LIN {X 0,Y 81.498,Z 212.955,A -85,B 0,C 180,E1 -29781.837,E2 -29781.837} C_VEL
LIN {X 0,Y 84.954,Z 223.328,A -85,B 0,C 180,E1 -29789.059,E2 -29789.059} C_VEL
LIN {X 0,Y 88.345,Z 233.499,A -85,B 0,C 180,E1 -29794.807,E2 -29794.807} C_VEL
LIN {X 0,Y 92.972,Z 247.732,A -85,B 0,C 180,E1 -29801.381,E2 -29801.381} C_VEL
LIN {X 0,Y 75.771,Z 322.387,A -85,B 0,C 180,E1 -29809.104,E2 -29809.104} C_VEL
LIN {X 0,Y 70.598,Z 340.758,A -85,B 0,C 180,E1 -29812.018,E2 -29812.018} C_VEL
LIN {X 0,Y 64.901,Z 358.077,A -85,B 0,C 180,E1 -29815.953,E2 -29815.953} C_VEL
LIN {X 0,Y 57.963,Z 376.296,A -85,B 0,C 180,E1 -29821.924,E2 -29821.924} C_VEL
LIN {X 0,Y 50.843,Z 393.773,A -85,B 0,C 180,E1 -29830.512,E2 -29830.512} C_VEL
LIN {X 0,Y 44.399,Z 410.254,A -85,B 0,C 180,E1 -29843.006,E2 -29843.006} C_VEL
LIN {X 0,Y 40.062,Z 424.851,A -85,B 0,C 180,E1 -29859.459,E2 -29859.459} C_VEL
LIN {X 0,Y 38.918,Z 435.167,A -85,B 0,C 180,E1 -29874.818,E2 -29874.818} C_VEL
LIN {X 0,Y 40.086,Z 444.149,A -85,B 0,C 180,E1 -29890.096,E2 -29890.096} C_VEL
LIN {X 0,Y 42.987,Z 451.752,A -85,B 0,C 180,E1 -29904.124,E2 -29904.124} C_VEL
LIN {X 0,Y 48.332,Z 459.273,A -85,B 0,C 180,E1 -29918.169,E2 -29918.169} C_VEL
LIN {X 0,Y 52.134,Z 462.9,A -85,B 0,C 180,E1 -29924.447,E2 -29924.447} C_VEL
LIN {X 0,Y 51.741,Z 462.795,A -85,B 0,C 180,E1 -29927.216,E2 -29927.216} C_VEL
LIN {X 0,Y 46.77,Z 457.154,A -85,B 0,C 180,E1 -29947.357,E2 -29947.357} C_VEL
LIN {X 0,Y 46.468,Z 455.688,A -85,B 0,C 180,E1 -29952.387,E2 -29952.387} C_VEL
LIN {X 0,Y 46.065,Z 453.922,A -85,B 0,C 180,E1 -29956.765,E2 -29956.765} C_VEL
LIN {X 0,Y 43.68,Z 447.526,A -85,B 0,C 180,E1 -29967.689,E2 -29967.689} C_VEL
LIN {X 0,Y 42.428,Z 436.729,A -85,B 0,C 180,E1 -29984.38,E2 -29984.38} C_VEL
LIN {X 0,Y 44.138,Z 425.938,A -85,B 0,C 180,E1 -29998.527,E2 -29998.527} C_VEL
LIN {X 0,Y 48.424,Z 412.157,A -85,B 0,C 180,E1 -30012.045,E2 -30012.045} C_VEL
LIN {X 0,Y 54.366,Z 397.007,A -85,B 0,C 180,E1 -30022.345,E2 -30022.345} C_VEL
LIN {X 0,Y 60.976,Z 380.581,A -85,B 0,C 180,E1 -30029.81,E2 -30029.81} C_VEL
LIN {X 0,Y 67.321,Z 363.42,A -85,B 0,C 180,E1 -30035.134,E2 -30035.134} C_VEL
LIN {X 0,Y 73.035,Z 346.162,A -85,B 0,C 180,E1 -30038.771,E2 -30038.771} C_VEL
LIN {X 0,Y 77.413,Z 329.485,A -85,B 0,C 180,E1 -30041.354,E2 -30041.354} C_VEL
LIN {X 0,Y 94.399,Z 256.118,A -85,B 0,C 180,E1 -30049.009,E2 -30049.009} C_VEL
LIN {X 0,Y 89.802,Z 238.607,A -85,B 0,C 180,E1 -30055.909,E2 -30055.909} C_VEL
LIN {X 0,Y 87.812,Z 231.246,A -85,B 0,C 180,E1 -30059.302,E2 -30059.302} C_VEL
LIN {X 0,Y 83.874,Z 219.706,A -85,B 0,C 180,E1 -30066.271,E2 -30066.271} C_VEL
LIN {X 0,Y 81.116,Z 211.549,A -85,B 0,C 180,E1 -30072.319,E2 -30072.319} C_VEL
LIN {X 0,Y 79.343,Z 206.703,A -85,B 0,C 180,E1 -30076.883,E2 -30076.883} C_VEL
LIN {X 0,Y 77.372,Z 202.569,A -85,B 0,C 180,E1 -30082.396,E2 -30082.396} C_VEL
LIN {X 0,Y 76.416,Z 200.778,A -85,B 0,C 180,E1 -30085.579,E2 -30085.579} C_VEL
LIN {X 0,Y 75.225,Z 198.037,A -85,B 0,C 180,E1 -30090.911,E2 -30090.911} C_VEL
LIN {X 0,Y 73.855,Z 194.358,A -85,B 0,C 180,E1 -30105.053,E2 -30105.053} C_VEL
LIN {X 0,Y 73.889,Z 194.326,A -85,B 0,C 180,E1 -30108.716,E2 -30108.716} C_VEL
LIN {X 0,Y 75.492,Z 198.537,A -85,B 0,C 180,E1 -30123.535,E2 -30123.535} C_VEL
LIN {X 0,Y 77.1,Z 201.774,A -85,B 0,C 180,E1 -30129.721,E2 -30129.721} C_VEL
LIN {X 0,Y 78.057,Z 203.875,A -85,B 0,C 180,E1 -30132.788,E2 -30132.788} C_VEL
LIN {X 0,Y 78.673,Z 206.225,A -85,B 0,C 180,E1 -30135,E2 -30135} C_VEL
LIN {X 0,Y 78.846,Z 209.414,A -85,B 0,C 180,E1 -30136.71,E2 -30136.71} C_VEL
LIN {X 0,Y 78.721,Z 219.635,A -85,B 0,C 180,E1 -30140.842,E2 -30140.842} C_VEL
LIN {X 0,Y 78.953,Z 221.239,A -85,B 0,C 180,E1 -30141.776,E2 -30141.776} C_VEL
LIN {X 0,Y 82.123,Z 231.652,A -85,B 0,C 180,E1 -30148.911,E2 -30148.911} C_VEL
LIN {X 0,Y 85.803,Z 243.983,A -85,B 0,C 180,E1 -30155.622,E2 -30155.622} C_VEL
LIN {X 0,Y 87.566,Z 249.754,A -85,B 0,C 180,E1 -30158.369,E2 -30158.369} C_VEL
LIN {X 0,Y 69.671,Z 323.884,A -85,B 0,C 180,E1 -30165.958,E2 -30165.958} C_VEL
LIN {X 0,Y 63.877,Z 343.313,A -85,B 0,C 180,E1 -30169.187,E2 -30169.187} C_VEL
LIN {X 0,Y 57.497,Z 361.158,A -85,B 0,C 180,E1 -30173.543,E2 -30173.543} C_VEL
LIN {X 0,Y 50.547,Z 378.063,A -85,B 0,C 180,E1 -30179.658,E2 -30179.658} C_VEL
LIN {X 0,Y 43.158,Z 395.148,A -85,B 0,C 180,E1 -30189.332,E2 -30189.332} C_VEL
LIN {X 0,Y 37.164,Z 409.779,A -85,B 0,C 180,E1 -30202.431,E2 -30202.431} C_VEL
LIN {X 0,Y 33.075,Z 423.75,A -85,B 0,C 180,E1 -30221.413,E2 -30221.413} C_VEL
LIN {X 0,Y 32.512,Z 434.151,A -85,B 0,C 180,E1 -30239.999,E2 -30239.999} C_VEL
LIN {X 0,Y 34.7,Z 443.052,A -85,B 0,C 180,E1 -30257.685,E2 -30257.685} C_VEL
LIN {X 0,Y 38.033,Z 449.406,A -85,B 0,C 180,E1 -30270.54,E2 -30270.54} C_VEL
LIN {X 0,Y 44.578,Z 457.016,A -85,B 0,C 180,E1 -30285.189,E2 -30285.189} C_VEL
LIN {X 0,Y 44.148,Z 456.848,A -85,B 0,C 180,E1 -30290.441,E2 -30290.441} C_VEL
LIN {X 0,Y 40.851,Z 451.711,A -85,B 0,C 180,E1 -30309.867,E2 -30309.867} C_VEL
LIN {X 0,Y 40.524,Z 450.826,A -85,B 0,C 180,E1 -30312.325,E2 -30312.325} C_VEL
LIN {X 0,Y 37.539,Z 444.264,A -85,B 0,C 180,E1 -30324.622,E2 -30324.622} C_VEL
LIN {X 0,Y 35.942,Z 433.295,A -85,B 0,C 180,E1 -30343.849,E2 -30343.849} C_VEL
LIN {X 0,Y 37.796,Z 421.958,A -85,B 0,C 180,E1 -30360.746,E2 -30360.746} C_VEL
LIN {X 0,Y 42.454,Z 408.36,A -85,B 0,C 180,E1 -30375.478,E2 -30375.478} C_VEL
LIN {X 0,Y 48.556,Z 393.763,A -85,B 0,C 180,E1 -30385.949,E2 -30385.949} C_VEL
LIN {X 0,Y 55.792,Z 376.675,A -85,B 0,C 180,E1 -30393.824,E2 -30393.824} C_VEL
LIN {X 0,Y 62.443,Z 359.243,A -85,B 0,C 180,E1 -30399.052,E2 -30399.052} C_VEL
LIN {X 0,Y 68.54,Z 340.751,A -85,B 0,C 180,E1 -30402.711,E2 -30402.711} C_VEL
LIN {X 0,Y 73.894,Z 319.765,A -85,B 0,C 180,E1 -30405.662,E2 -30405.662} C_VEL
LIN {X 0,Y 88.85,Z 257.627,A -85,B 0,C 180,E1 -30411.928,E2 -30411.928} C_VEL
LIN {X 0,Y 84.552,Z 239.719,A -85,B 0,C 180,E1 -30419.612,E2 -30419.612} C_VEL
LIN {X 0,Y 82.874,Z 233.486,A -85,B 0,C 180,E1 -30422.934,E2 -30422.934} C_VEL
LIN {X 0,Y 79.607,Z 222.985,A -85,B 0,C 180,E1 -30429.922,E2 -30429.922} C_VEL
LIN {X 0,Y 77.751,Z 216.749,A -85,B 0,C 180,E1 -30434.853,E2 -30434.853} C_VEL
LIN {X 0,Y 76.283,Z 212.249,A -85,B 0,C 180,E1 -30439.302,E2 -30439.302} C_VEL
LIN {X 0,Y 74.59,Z 208.154,A -85,B 0,C 180,E1 -30445.095,E2 -30445.095} C_VEL
LIN {X 0,Y 72.897,Z 204.473,A -85,B 0,C 180,E1 -30453.029,E2 -30453.029} C_VEL
LIN {X 0,Y 72.031,Z 201.284,A -85,B 0,C 180,E1 -30465.368,E2 -30465.368} C_VEL
LIN {X 0,Y 72.043,Z 201.372,A -85,B 0,C 180,E1 -30468.824,E2 -30468.824} C_VEL
LIN {X 0,Y 73.299,Z 205.017,A -85,B 0,C 180,E1 -30482.109,E2 -30482.109} C_VEL
LIN {X 0,Y 74.607,Z 208.12,A -85,B 0,C 180,E1 -30488.111,E2 -30488.111} C_VEL
LIN {X 0,Y 76.025,Z 211.531,A -85,B 0,C 180,E1 -30493.009,E2 -30493.009} C_VEL
LIN {X 0,Y 78.067,Z 218.145,A -85,B 0,C 180,E1 -30499.326,E2 -30499.326} C_VEL
LIN {X 0,Y 78.953,Z 221.239,A -85,B 0,C 180,E1 -30501.776,E2 -30501.776} C_VEL
LIN {X 0,Y 79.615,Z 225.956,A -85,B 0,C 180,E1 -30504.324,E2 -30504.324} C_VEL
LIN {X 0,Y 80.263,Z 241.827,A -85,B 0,C 180,E1 -30510.295,E2 -30510.295} C_VEL
LIN {X 0,Y 80.995,Z 246.877,A -85,B 0,C 180,E1 -30512.491,E2 -30512.491} C_VEL
LIN {X 0,Y 81.406,Z 248.447,A -85,B 0,C 180,E1 -30513.301,E2 -30513.301} C_VEL
LIN {X 0,Y 82.262,Z 251.953,A -85,B 0,C 180,E1 -30515.004,E2 -30515.004} C_VEL
LIN {X 0,Y 63.862,Z 324.871,A -85,B 0,C 180,E1 -30522.233,E2 -30522.233} C_VEL
LIN {X 0,Y 57.856,Z 343.978,A -85,B 0,C 180,E1 -30525.374,E2 -30525.374} C_VEL
LIN {X 0,Y 51.294,Z 361.232,A -85,B 0,C 180,E1 -30529.611,E2 -30529.611} C_VEL
LIN {X 0,Y 43.262,Z 379.609,A -85,B 0,C 180,E1 -30536.683,E2 -30536.683} C_VEL
LIN {X 0,Y 36.438,Z 394.333,A -85,B 0,C 180,E1 -30546.02,E2 -30546.02} C_VEL
LIN {X 0,Y 30.332,Z 408.259,A -85,B 0,C 180,E1 -30560.416,E2 -30560.416} C_VEL
LIN {X 0,Y 26.502,Z 420.672,A -85,B 0,C 180,E1 -30580.639,E2 -30580.639} C_VEL
LIN {X 0,Y 26.221,Z 431.325,A -85,B 0,C 180,E1 -30603.84,E2 -30603.84} C_VEL
LIN {X 0,Y 29.373,Z 440.52,A -85,B 0,C 180,E1 -30624.752,E2 -30624.752} C_VEL
LIN {X 0,Y 33.712,Z 446.988,A -85,B 0,C 180,E1 -30638.711,E2 -30638.711} C_VEL
LIN {X 0,Y 37.995,Z 451.483,A -85,B 0,C 180,E1 -30647.719,E2 -30647.719} C_VEL
LIN {X 0,Y 36.96,Z 450.439,A -85,B 0,C 180,E1 -30655.21,E2 -30655.21} C_VEL
LIN {X 0,Y 35.36,Z 447.641,A -85,B 0,C 180,E1 -30666.569,E2 -30666.569} C_VEL
LIN {X 0,Y 31.641,Z 440.824,A -85,B 0,C 180,E1 -30680.402,E2 -30680.402} C_VEL
LIN {X 0,Y 29.502,Z 429.42,A -85,B 0,C 180,E1 -30703.772,E2 -30703.772} C_VEL
LIN {X 0,Y 31.926,Z 416.835,A -85,B 0,C 180,E1 -30725.29,E2 -30725.29} C_VEL
LIN {X 0,Y 36.71,Z 404.254,A -85,B 0,C 180,E1 -30739.965,E2 -30739.965} C_VEL
LIN {X 0,Y 43.547,Z 389.197,A -85,B 0,C 180,E1 -30751.044,E2 -30751.044} C_VEL
LIN {X 0,Y 50.212,Z 374.114,A -85,B 0,C 180,E1 -30758.001,E2 -30758.001} C_VEL
LIN {X 0,Y 56.948,Z 357.238,A -85,B 0,C 180,E1 -30763.007,E2 -30763.007} C_VEL
LIN {X 0,Y 63.045,Z 339.479,A -85,B 0,C 180,E1 -30766.464,E2 -30766.464} C_VEL
LIN {X 0,Y 68.889,Z 317.321,A -85,B 0,C 180,E1 -30769.514,E2 -30769.514} C_VEL
LIN {X 0,Y 83.47,Z 259.201,A -85,B 0,C 180,E1 -30775.171,E2 -30775.171} C_VEL
LIN {X 0,Y 79.716,Z 241.586,A -85,B 0,C 180,E1 -30783.392,E2 -30783.392} C_VEL
LIN {X 0,Y 76.894,Z 231.111,A -85,B 0,C 180,E1 -30790.163,E2 -30790.163} C_VEL
LIN {X 0,Y 74.595,Z 222.191,A -85,B 0,C 180,E1 -30797.318,E2 -30797.318} C_VEL
LIN {X 0,Y 73.264,Z 217.466,A -85,B 0,C 180,E1 -30802.305,E2 -30802.305} C_VEL
LIN {X 0,Y 71.905,Z 213.883,A -85,B 0,C 180,E1 -30807.925,E2 -30807.925} C_VEL
LIN {X 0,Y 70.846,Z 211.124,A -85,B 0,C 180,E1 -30814.114,E2 -30814.114} C_VEL
LIN {X 0,Y 70.211,Z 208.208,A -85,B 0,C 180,E1 -30825.523,E2 -30825.523} C_VEL
LIN {X 0,Y 70.221,Z 208.256,A -85,B 0,C 180,E1 -30828.23,E2 -30828.23} C_VEL
LIN {X 0,Y 71.155,Z 211.686,A -85,B 0,C 180,E1 -30840.895,E2 -30840.895} C_VEL
LIN {X 0,Y 72.215,Z 214.562,A -85,B 0,C 180,E1 -30846.57,E2 -30846.57} C_VEL
LIN {X 0,Y 73.247,Z 217.36,A -85,B 0,C 180,E1 -30850.739,E2 -30850.739} C_VEL
LIN {X 0,Y 74.852,Z 223.675,A -85,B 0,C 180,E1 -30856.974,E2 -30856.974} C_VEL
LIN {X 0,Y 77.129,Z 232.534,A -85,B 0,C 180,E1 -30863.796,E2 -30863.796} C_VEL
LIN {X 0,Y 79.834,Z 242.675,A -85,B 0,C 180,E1 -30870.161,E2 -30870.161} C_VEL
LIN {X 0,Y 81.406,Z 248.447,A -85,B 0,C 180,E1 -30873.301,E2 -30873.301} C_VEL
LIN {X 0,Y 81.47,Z 250.935,A -85,B 0,C 180,E1 -30874.067,E2 -30874.067} C_VEL
LIN {X 0,Y 80.482,Z 254.277,A -85,B 0,C 180,E1 -30874.212,E2 -30874.212} C_VEL
LIN {X 0,Y 78.716,Z 257.792,A -85,B 0,C 180,E1 -30873.757,E2 -30873.757} C_VEL
LIN {X 0,Y 75.065,Z 264.078,A -85,B 0,C 180,E1 -30872.425,E2 -30872.425} C_VEL
LIN {X 0,Y 73.483,Z 268.168,A -85,B 0,C 180,E1 -30872.25,E2 -30872.25} C_VEL
LIN {X 0,Y 58.17,Z 326.394,A -85,B 0,C 180,E1 -30877.95,E2 -30877.95} C_VEL
LIN {X 0,Y 51.475,Z 346.175,A -85,B 0,C 180,E1 -30881.087,E2 -30881.087} C_VEL
LIN {X 0,Y 44.606,Z 362.93,A -85,B 0,C 180,E1 -30885.194,E2 -30885.194} C_VEL
LIN {X 0,Y 36.94,Z 379.442,A -85,B 0,C 180,E1 -30891.785,E2 -30891.785} C_VEL
LIN {X 0,Y 29.62,Z 393.953,A -85,B 0,C 180,E1 -30901.804,E2 -30901.804} C_VEL
LIN {X 0,Y 22.99,Z 407.945,A -85,B 0,C 180,E1 -30919.487,E2 -30919.487} C_VEL
LIN {X 0,Y 19.469,Z 421.233,A -85,B 0,C 180,E1 -30949.599,E2 -30949.599} C_VEL
LIN {X 0,Y 21.34,Z 431.669,A -85,B 0,C 180,E1 -30979.226,E2 -30979.226} C_VEL
LIN {X 0,Y 25.791,Z 439.167,A -85,B 0,C 180,E1 -30997.814,E2 -30997.814} C_VEL
LIN {X 0,Y 30.99,Z 444.961,A -85,B 0,C 180,E1 -31010.119,E2 -31010.119} C_VEL
LIN {X 0,Y 31.163,Z 444.964,A -85,B 0,C 180,E1 -31015.671,E2 -31015.671} C_VEL
LIN {X 0,Y 29.715,Z 443.029,A -85,B 0,C 180,E1 -31021.759,E2 -31021.759} C_VEL
LIN {X 0,Y 24.59,Z 434.111,A -85,B 0,C 180,E1 -31041.773,E2 -31041.773} C_VEL
LIN {X 0,Y 23.392,Z 422.203,A -85,B 0,C 180,E1 -31071.001,E2 -31071.001} C_VEL
LIN {X 0,Y 26.818,Z 410.267,A -85,B 0,C 180,E1 -31093.452,E2 -31093.452} C_VEL
LIN {X 0,Y 34.059,Z 394.497,A -85,B 0,C 180,E1 -31110.823,E2 -31110.823} C_VEL
LIN {X 0,Y 41.837,Z 378.355,A -85,B 0,C 180,E1 -31120.37,E2 -31120.37} C_VEL
LIN {X 0,Y 48.892,Z 362.291,A -85,B 0,C 180,E1 -31125.974,E2 -31125.974} C_VEL
LIN {X 0,Y 55.357,Z 345.454,A -85,B 0,C 180,E1 -31129.682,E2 -31129.682} C_VEL
LIN {X 0,Y 60.205,Z 329.929,A -85,B 0,C 180,E1 -31132.059,E2 -31132.059} C_VEL
LIN {X 0,Y 78.298,Z 261.003,A -85,B 0,C 180,E1 -31138.742,E2 -31138.742} C_VEL
LIN {X 0,Y 75.44,Z 244.997,A -85,B 0,C 180,E1 -31146.752,E2 -31146.752} C_VEL
LIN {X 0,Y 72.844,Z 233.903,A -85,B 0,C 180,E1 -31154.626,E2 -31154.626} C_VEL
LIN {X 0,Y 71.443,Z 227.302,A -85,B 0,C 180,E1 -31160.319,E2 -31160.319} C_VEL
LIN {X 0,Y 70.488,Z 223.026,A -85,B 0,C 180,E1 -31165.046,E2 -31165.046} C_VEL
LIN {X 0,Y 69.52,Z 220.101,A -85,B 0,C 180,E1 -31170.096,E2 -31170.096} C_VEL
LIN {X 0,Y 68.752,Z 217.733,A -85,B 0,C 180,E1 -31175.67,E2 -31175.67} C_VEL
LIN {X 0,Y 68.405,Z 215.075,A -85,B 0,C 180,E1 -31185.988,E2 -31185.988} C_VEL
LIN {X 0,Y 68.366,Z 215.322,A -85,B 0,C 180,E1 -31188.129,E2 -31188.129} C_VEL
LIN {X 0,Y 69.058,Z 218.343,A -85,B 0,C 180,E1 -31199.67,E2 -31199.67} C_VEL
LIN {X 0,Y 69.863,Z 220.948,A -85,B 0,C 180,E1 -31204.875,E2 -31204.875} C_VEL
LIN {X 0,Y 70.531,Z 223.328,A -85,B 0,C 180,E1 -31208.444,E2 -31208.444} C_VEL
LIN {X 0,Y 71.661,Z 228.84,A -85,B 0,C 180,E1 -31214.074,E2 -31214.074} C_VEL
LIN {X 0,Y 73.674,Z 238.195,A -85,B 0,C 180,E1 -31221.577,E2 -31221.577} C_VEL
LIN {X 0,Y 76.068,Z 248.61,A -85,B 0,C 180,E1 -31228.292,E2 -31228.292} C_VEL
LIN {X 0,Y 77.271,Z 253.53,A -85,B 0,C 180,E1 -31231.143,E2 -31231.143} C_VEL
LIN {X 0,Y 73.483,Z 268.168,A -85,B 0,C 180,E1 -31232.25,E2 -31232.25} C_VEL
LIN {X 0,Y 71.584,Z 273.769,A -85,B 0,C 180,E1 -31232.259,E2 -31232.259} C_VEL
LIN {X 0,Y 63.137,Z 291.505,A -85,B 0,C 180,E1 -31229.752,E2 -31229.752} C_VEL
LIN {X 0,Y 61.295,Z 297.107,A -85,B 0,C 180,E1 -31229.819,E2 -31229.819} C_VEL
LIN {X 0,Y 52.772,Z 327.736,A -85,B 0,C 180,E1 -31232.756,E2 -31232.756} C_VEL
LIN {X 0,Y 45.893,Z 347.022,A -85,B 0,C 180,E1 -31235.488,E2 -31235.488} C_VEL
LIN {X 0,Y 39.117,Z 362.687,A -85,B 0,C 180,E1 -31238.818,E2 -31238.818} C_VEL
LIN {X 0,Y 30.858,Z 379.265,A -85,B 0,C 180,E1 -31245.036,E2 -31245.036} C_VEL
LIN {X 0,Y 23.243,Z 393.132,A -85,B 0,C 180,E1 -31254.886,E2 -31254.886} C_VEL
LIN {X 0,Y 16.222,Z 406.413,A -85,B 0,C 180,E1 -31275.246,E2 -31275.246} C_VEL
LIN {X 0,Y 13.011,Z 417.854,A -85,B 0,C 180,E1 -31312.236,E2 -31312.236} C_VEL
LIN {X 0,Y 16.806,Z 429.205,A -85,B 0,C 180,E1 -31353.985,E2 -31353.985} C_VEL
LIN {X 0,Y 22.538,Z 436.29,A -85,B 0,C 180,E1 -31371.233,E2 -31371.233} C_VEL
LIN {X 0,Y 24.332,Z 438.093,A -85,B 0,C 180,E1 -31374.7,E2 -31374.7} C_VEL
LIN {X 0,Y 18.171,Z 428.588,A -85,B 0,C 180,E1 -31398.834,E2 -31398.834} C_VEL
LIN {X 0,Y 17.126,Z 417.498,A -85,B 0,C 180,E1 -31434.211,E2 -31434.211} C_VEL
LIN {X 0,Y 21.918,Z 404.442,A -85,B 0,C 180,E1 -31463.266,E2 -31463.266} C_VEL
LIN {X 0,Y 29.971,Z 388.986,A -85,B 0,C 180,E1 -31479.688,E2 -31479.688} C_VEL
LIN {X 0,Y 38.535,Z 372.161,A -85,B 0,C 180,E1 -31488.199,E2 -31488.199} C_VEL
LIN {X 0,Y 46.026,Z 355.278,A -85,B 0,C 180,E1 -31492.946,E2 -31492.946} C_VEL
LIN {X 0,Y 52.408,Z 338.304,A -85,B 0,C 180,E1 -31495.781,E2 -31495.781} C_VEL
LIN {X 0,Y 58.444,Z 317.586,A -85,B 0,C 180,E1 -31498.281,E2 -31498.281} C_VEL
LIN {X 0,Y 73.366,Z 262.564,A -85,B 0,C 180,E1 -31502.8,E2 -31502.8} C_VEL
LIN {X 0,Y 71.336,Z 248.584,A -85,B 0,C 180,E1 -31510.377,E2 -31510.377} C_VEL
LIN {X 0,Y 69.422,Z 238.447,A -85,B 0,C 180,E1 -31518.046,E2 -31518.046} C_VEL
LIN {X 0,Y 68.463,Z 232.374,A -85,B 0,C 180,E1 -31523.615,E2 -31523.615} C_VEL
LIN {X 0,Y 67.836,Z 228.542,A -85,B 0,C 180,E1 -31528.054,E2 -31528.054} C_VEL
LIN {X 0,Y 67.061,Z 225.852,A -85,B 0,C 180,E1 -31533.357,E2 -31533.357} C_VEL
LIN {X 0,Y 66.678,Z 224.232,A -85,B 0,C 180,E1 -31537.605,E2 -31537.605} C_VEL
LIN {X 0,Y 66.587,Z 221.962,A -85,B 0,C 180,E1 -31546.683,E2 -31546.683} C_VEL
LIN {X 0,Y 66.981,Z 224.979,A -85,B 0,C 180,E1 -31558.361,E2 -31558.361} C_VEL
LIN {X 0,Y 67.626,Z 227.665,A -85,B 0,C 180,E1 -31563.667,E2 -31563.667} C_VEL
LIN {X 0,Y 68.067,Z 230.116,A -85,B 0,C 180,E1 -31566.977,E2 -31566.977} C_VEL
LIN {X 0,Y 68.889,Z 235.69,A -85,B 0,C 180,E1 -31572.491,E2 -31572.491} C_VEL
LIN {X 0,Y 70.748,Z 246.249,A -85,B 0,C 180,E1 -31580.895,E2 -31580.895} C_VEL
LIN {X 0,Y 72.502,Z 255.356,A -85,B 0,C 180,E1 -31586.805,E2 -31586.805} C_VEL
LIN {X 0,Y 61.295,Z 297.107,A -85,B 0,C 180,E1 -31589.819,E2 -31589.819} C_VEL
LIN {X 0,Y 59.487,Z 302.71,A -85,B 0,C 180,E1 -31589.938,E2 -31589.938} C_VEL
LIN {X 0,Y 55.38,Z 311.602,A -85,B 0,C 180,E1 -31588.592,E2 -31588.592} C_VEL
LIN {X 0,Y 51.893,Z 318.639,A -85,B 0,C 180,E1 -31587.019,E2 -31587.019} C_VEL
LIN {X 0,Y 49.543,Z 324.083,A -85,B 0,C 180,E1 -31586.339,E2 -31586.339} C_VEL
LIN {X 0,Y 48.864,Z 325.949,A -85,B 0,C 180,E1 -31586.313,E2 -31586.313} C_VEL
LIN {X 0,Y 41.75,Z 345.532,A -85,B 0,C 180,E1 -31588.159,E2 -31588.159} C_VEL
LIN {X 0,Y 34.351,Z 362.021,A -85,B 0,C 180,E1 -31590.591,E2 -31590.591} C_VEL
LIN {X 0,Y 26.444,Z 377.134,A -85,B 0,C 180,E1 -31594.677,E2 -31594.677} C_VEL
LIN {X 0,Y 17.999,Z 391.315,A -85,B 0,C 180,E1 -31602.519,E2 -31602.519} C_VEL
LIN {X 0,Y 9.678,Z 404.758,A -85,B 0,C 180,E1 -31625.215,E2 -31625.215} C_VEL
LIN {X 0,Y 7.541,Z 417.333,A -85,B 0,C 180,E1 -31701.15,E2 -31701.15} C_VEL
LIN {X 0,Y 12.251,Z 424.401,A -85,B 0,C 180,E1 -31731.383,E2 -31731.383} C_VEL
LIN {X 0,Y 14.01,Z 426.262,A -85,B 0,C 180,E1 -31739.868,E2 -31739.868} C_VEL
LIN {X 0,Y 10.531,Z 415.131,A -85,B 0,C 180,E1 -31789.465,E2 -31789.465} C_VEL
LIN {X 0,Y 15.89,Z 401.944,A -85,B 0,C 180,E1 -31832.163,E2 -31832.163} C_VEL
LIN {X 0,Y 25.051,Z 386.307,A -85,B 0,C 180,E1 -31849.026,E2 -31849.026} C_VEL
LIN {X 0,Y 33.467,Z 370.827,A -85,B 0,C 180,E1 -31855.827,E2 -31855.827} C_VEL
LIN {X 0,Y 41.272,Z 354.005,A -85,B 0,C 180,E1 -31859.677,E2 -31859.677} C_VEL
LIN {X 0,Y 48.254,Z 335.987,A -85,B 0,C 180,E1 -31862.004,E2 -31862.004} C_VEL
LIN {X 0,Y 55.727,Z 310.631,A -85,B 0,C 180,E1 -31864.427,E2 -31864.427} C_VEL
LIN {X 0,Y 68.756,Z 263.901,A -85,B 0,C 180,E1 -31867.476,E2 -31867.476} C_VEL
LIN {X 0,Y 67.497,Z 252.062,A -85,B 0,C 180,E1 -31874.474,E2 -31874.474} C_VEL
LIN {X 0,Y 66.161,Z 242.343,A -85,B 0,C 180,E1 -31882.421,E2 -31882.421} C_VEL
LIN {X 0,Y 65.638,Z 236.892,A -85,B 0,C 180,E1 -31887.719,E2 -31887.719} C_VEL
LIN {X 0,Y 65.325,Z 234.122,A -85,B 0,C 180,E1 -31891.344,E2 -31891.344} C_VEL
LIN {X 0,Y 64.776,Z 231.045,A -85,B 0,C 180,E1 -31898.142,E2 -31898.142} C_VEL
LIN {X 0,Y 64.653,Z 229.23,A -85,B 0,C 180,E1 -31905.508,E2 -31905.508} C_VEL
LIN {X 0,Y 64.602,Z 229.559,A -85,B 0,C 180,E1 -31908.702,E2 -31908.702} C_VEL
LIN {X 0,Y 64.935,Z 231.616,A -85,B 0,C 180,E1 -31916.954,E2 -31916.954} C_VEL
LIN {X 0,Y 65.366,Z 234.254,A -85,B 0,C 180,E1 -31922.135,E2 -31922.135} C_VEL
LIN {X 0,Y 65.753,Z 238.976,A -85,B 0,C 180,E1 -31927.381,E2 -31927.381} C_VEL
LIN {X 0,Y 66.723,Z 247.446,A -85,B 0,C 180,E1 -31934.884,E2 -31934.884} C_VEL
LIN {X 0,Y 68.135,Z 257.55,A -85,B 0,C 180,E1 -31942.119,E2 -31942.119} C_VEL
LIN {X 0,Y 49.302,Z 324.593,A -85,B 0,C 180,E1 -31946.245,E2 -31946.245} C_VEL
LIN {X 0,Y 48.864,Z 325.949,A -85,B 0,C 180,E1 -31946.313,E2 -31946.313} C_VEL
LIN {X 0,Y 46.576,Z 331.396,A -85,B 0,C 180,E1 -31945.881,E2 -31945.881} C_VEL
LIN {X 0,Y 36.859,Z 348.267,A -85,B 0,C 180,E1 -31940.472,E2 -31940.472} C_VEL
LIN {X 0,Y 34.184,Z 353.548,A -85,B 0,C 180,E1 -31939.872,E2 -31939.872} C_VEL
LIN {X 0,Y 24.927,Z 371.851,A -85,B 0,C 180,E1 -31940.694,E2 -31940.694} C_VEL
LIN {X 0,Y 15.971,Z 386.656,A -85,B 0,C 180,E1 -31941.945,E2 -31941.945} C_VEL
LIN {X 0,Y 6.086,Z 400.733,A -85,B 0,C 180,E1 -31944.988,E2 -31944.988} C_VEL
LIN {X 0,Y 2.804,Z 411.61,A -85,B 0,C 180,E1 -32116.008,E2 -32116.008} C_VEL
LIN {X 0,Y 4.284,Z 412.637,A -85,B 0,C 180,E1 -32129.938,E2 -32129.938} C_VEL
LIN {X 0,Y 10.558,Z 399.472,A -85,B 0,C 180,E1 -32210.178,E2 -32210.178} C_VEL
LIN {X 0,Y 21.097,Z 383.497,A -85,B 0,C 180,E1 -32222.38,E2 -32222.38} C_VEL
LIN {X 0,Y 30.038,Z 367.651,A -85,B 0,C 180,E1 -32226.161,E2 -32226.161} C_VEL
LIN {X 0,Y 38.556,Z 349.647,A -85,B 0,C 180,E1 -32228.171,E2 -32228.171} C_VEL
LIN {X 0,Y 44.755,Z 333.585,A -85,B 0,C 180,E1 -32229.217,E2 -32229.217} C_VEL
LIN {X 0,Y 54.858,Z 299.342,A -85,B 0,C 180,E1 -32231.251,E2 -32231.251} C_VEL
LIN {X 0,Y 64.581,Z 265.574,A -85,B 0,C 180,E1 -32232.572,E2 -32232.572} C_VEL
LIN {X 0,Y 64.013,Z 256.06,A -85,B 0,C 180,E1 -32238.59,E2 -32238.59} C_VEL
LIN {X 0,Y 63.258,Z 246.822,A -85,B 0,C 180,E1 -32246.599,E2 -32246.599} C_VEL
LIN {X 0,Y 63.138,Z 242.277,A -85,B 0,C 180,E1 -32251.178,E2 -32251.178} C_VEL
LIN {X 0,Y 63.013,Z 240.026,A -85,B 0,C 180,E1 -32254.28,E2 -32254.28} C_VEL
LIN {X 0,Y 62.756,Z 237.509,A -85,B 0,C 180,E1 -32260.417,E2 -32260.417} C_VEL
LIN {X 0,Y 62.749,Z 236.433,A -85,B 0,C 180,E1 -32264.775,E2 -32264.775} C_VEL
LIN {X 0,Y 62.76,Z 236.439,A -85,B 0,C 180,E1 -32268.194,E2 -32268.194} C_VEL
LIN {X 0,Y 62.887,Z 238.128,A -85,B 0,C 180,E1 -32275.139,E2 -32275.139} C_VEL
LIN {X 0,Y 63.066,Z 240.606,A -85,B 0,C 180,E1 -32279.816,E2 -32279.816} C_VEL
LIN {X 0,Y 63.158,Z 245.274,A -85,B 0,C 180,E1 -32284.874,E2 -32284.874} C_VEL
LIN {X 0,Y 63.783,Z 255.068,A -85,B 0,C 180,E1 -32293.482,E2 -32293.482} C_VEL
LIN {X 0,Y 64.203,Z 259.429,A -85,B 0,C 180,E1 -32296.764,E2 -32296.764} C_VEL
LIN {X 0,Y 45.425,Z 324.53,A -85,B 0,C 180,E1 -32298.963,E2 -32298.963} C_VEL
LIN {X 0,Y 38.513,Z 343.533,A -85,B 0,C 180,E1 -32299.493,E2 -32299.493} C_VEL
LIN {X 0,Y 34.184,Z 353.548,A -85,B 0,C 180,E1 -32299.872,E2 -32299.872} C_VEL
LIN {X 0,Y 31.41,Z 358.737,A -85,B 0,C 180,E1 -32298.964,E2 -32298.964} C_VEL
LIN {X 0,Y 26.022,Z 366.614,A -85,B 0,C 180,E1 -32293.505,E2 -32293.505} C_VEL
LIN {X 0,Y 20.73,Z 374.332,A -85,B 0,C 180,E1 -32284.994,E2 -32284.994} C_VEL
LIN {X 0,Y 17.744,Z 379.284,A -85,B 0,C 180,E1 -32280.873,E2 -32280.873} C_VEL
LIN {X 0,Y 8.531,Z 395.054,A -85,B 0,C 180,E1 -32257.823,E2 -32257.823} C_VEL
LIN {X 0,Y 8.003,Z 396.454,A -85,B 0,C 180,E1 -32248.652,E2 -32248.652} C_VEL
LIN {X 0,Y 17.679,Z 382.149,A -85,B 0,C 180,E1 -32240.547,E2 -32240.547} C_VEL
LIN {X 0,Y 26.872,Z 366.102,A -85,B 0,C 180,E1 -32238.58,E2 -32238.58} C_VEL
LIN {X 0,Y 35.512,Z 347.891,A -85,B 0,C 180,E1 -32237.774,E2 -32237.774} C_VEL
LIN {X 0,Y 41.956,Z 331.057,A -85,B 0,C 180,E1 -32237.49,E2 -32237.49} C_VEL
LIN {X 0,Y 60.898,Z 266.895,A -85,B 0,C 180,E1 -32238.455,E2 -32238.455} C_VEL
LIN {X 0,Y 60.794,Z 259.913,A -85,B 0,C 180,E1 -32243.26,E2 -32243.26} C_VEL
LIN {X 0,Y 60.671,Z 251.58,A -85,B 0,C 180,E1 -32250.869,E2 -32250.869} C_VEL
LIN {X 0,Y 60.836,Z 247.366,A -85,B 0,C 180,E1 -32255.284,E2 -32255.284} C_VEL
LIN {X 0,Y 60.888,Z 245.695,A -85,B 0,C 180,E1 -32257.842,E2 -32257.842} C_VEL
LIN {X 0,Y 60.839,Z 243.904,A -85,B 0,C 180,E1 -32262.918,E2 -32262.918} C_VEL
LIN {X 0,Y 60.934,Z 243.222,A -85,B 0,C 180,E1 -32267.039,E2 -32267.039} C_VEL
LIN {X 0,Y 60.907,Z 244.764,A -85,B 0,C 180,E1 -32273.632,E2 -32273.632} C_VEL
LIN {X 0,Y 60.872,Z 246.811,A -85,B 0,C 180,E1 -32277.077,E2 -32277.077} C_VEL
LIN {X 0,Y 60.594,Z 254.331,A -85,B 0,C 180,E1 -32284.716,E2 -32284.716} C_VEL
LIN {X 0,Y 60.726,Z 261.462,A -85,B 0,C 180,E1 -32290.782,E2 -32290.782} C_VEL
LIN {X 0,Y 42.623,Z 323.56,A -85,B 0,C 180,E1 -32290.592,E2 -32290.592} C_VEL
LIN {X 0,Y 35.354,Z 343.612,A -85,B 0,C 180,E1 -32289.392,E2 -32289.392} C_VEL
LIN {X 0,Y 27.643,Z 360.761,A -85,B 0,C 180,E1 -32287.168,E2 -32287.168} C_VEL
LIN {X 0,Y 18.903,Z 377.237,A -85,B 0,C 180,E1 -32282.011,E2 -32282.011} C_VEL
LIN {X 0,Y 17.744,Z 379.284,A -85,B 0,C 180,E1 -32280.873,E2 -32280.873} C_VEL
LIN {X 0,Y 17.41,Z 379.54,A -85,B 0,C 180,E1 -32277.427,E2 -32277.427} C_VEL
LIN {X 0,Y 17.723,Z 378.51,A -85,B 0,C 180,E1 -32271.303,E2 -32271.303} C_VEL
LIN {X 0,Y 19.177,Z 375.641,A -85,B 0,C 180,E1 -32263.871,E2 -32263.871} C_VEL
LIN {X 0,Y 22.597,Z 369.315,A -85,B 0,C 180,E1 -32256.595,E2 -32256.595} C_VEL
LIN {X 0,Y 26.038,Z 362.676,A -85,B 0,C 180,E1 -32252.757,E2 -32252.757} C_VEL
LIN {X 0,Y 33.536,Z 346.062,A -85,B 0,C 180,E1 -32248.668,E2 -32248.668} C_VEL
LIN {X 0,Y 39.788,Z 329.241,A -85,B 0,C 180,E1 -32246.723,E2 -32246.723} C_VEL
LIN {X 0,Y 57.752,Z 268.524,A -85,B 0,C 180,E1 -32244.844,E2 -32244.844} C_VEL
LIN {X 0,Y 57.994,Z 263.563,A -85,B 0,C 180,E1 -32248.545,E2 -32248.545} C_VEL
LIN {X 0,Y 58.468,Z 255.502,A -85,B 0,C 180,E1 -32256.297,E2 -32256.297} C_VEL
LIN {X 0,Y 58.896,Z 252.058,A -85,B 0,C 180,E1 -32260.132,E2 -32260.132} C_VEL
LIN {X 0,Y 59.016,Z 250.443,A -85,B 0,C 180,E1 -32264.979,E2 -32264.979} C_VEL
LIN {X 0,Y 59.036,Z 250.48,A -85,B 0,C 180,E1 -32268.695,E2 -32268.695} C_VEL
LIN {X 0,Y 58.936,Z 251.594,A -85,B 0,C 180,E1 -32272.208,E2 -32272.208} C_VEL
LIN {X 0,Y 58.432,Z 255.725,A -85,B 0,C 180,E1 -32276.93,E2 -32276.93} C_VEL
LIN {X 0,Y 57.898,Z 263.443,A -85,B 0,C 180,E1 -32284.188,E2 -32284.188} C_VEL
LIN {X 0,Y 40.539,Z 323.282,A -85,B 0,C 180,E1 -32281.194,E2 -32281.194} C_VEL
LIN {X 0,Y 33.674,Z 342.918,A -85,B 0,C 180,E1 -32277.983,E2 -32277.983} C_VEL
LIN {X 0,Y 26.612,Z 359.794,A -85,B 0,C 180,E1 -32272.401,E2 -32272.401} C_VEL
LIN {X 0,Y 20.397,Z 373.246,A -85,B 0,C 180,E1 -32263.563,E2 -32263.563} C_VEL
LIN {X 0,Y 20.133,Z 374.201,A -85,B 0,C 180,E1 -32258.215,E2 -32258.215} C_VEL
LIN {X 0,Y 26.038,Z 362.676,A -85,B 0,C 180,E1 -32252.757,E2 -32252.757} C_VEL
LIN {X 0,Y 28.441,Z 357.391,A -85,B 0,C 180,E1 -32252.376,E2 -32252.376} C_VEL
LIN {X 0,Y 31.801,Z 348.302,A -85,B 0,C 180,E1 -32255.081,E2 -32255.081} C_VEL
LIN {X 0,Y 34.307,Z 340.757,A -85,B 0,C 180,E1 -32257.381,E2 -32257.381} C_VEL
LIN {X 0,Y 36.189,Z 335.009,A -85,B 0,C 180,E1 -32257.856,E2 -32257.856} C_VEL
LIN {X 0,Y 36.834,Z 333.088,A -85,B 0,C 180,E1 -32257.641,E2 -32257.641} C_VEL
LIN {X 0,Y 44.464,Z 307.717,A -85,B 0,C 180,E1 -32254.538,E2 -32254.538} C_VEL
LIN {X 0,Y 55.307,Z 270.163,A -85,B 0,C 180,E1 -32251.814,E2 -32251.814} C_VEL
LIN {X 0,Y 56.188,Z 262.809,A -85,B 0,C 180,E1 -32258.471,E2 -32258.471} C_VEL
LIN {X 0,Y 57.032,Z 257.993,A -85,B 0,C 180,E1 -32263.681,E2 -32263.681} C_VEL
LIN {X 0,Y 57.192,Z 257.207,A -85,B 0,C 180,E1 -32266.176,E2 -32266.176} C_VEL
LIN {X 0,Y 57.151,Z 257.518,A -85,B 0,C 180,E1 -32268.723,E2 -32268.723} C_VEL
LIN {X 0,Y 55.848,Z 264.924,A -85,B 0,C 180,E1 -32276.444,E2 -32276.444} C_VEL
LIN {X 0,Y 55.769,Z 265.56,A -85,B 0,C 180,E1 -32277.027,E2 -32277.027} C_VEL
LIN {X 0,Y 39.937,Z 321.638,A -85,B 0,C 180,E1 -32271.344,E2 -32271.344} C_VEL
LIN {X 0,Y 33.951,Z 340.526,A -85,B 0,C 180,E1 -32266.431,E2 -32266.431} C_VEL
LIN {X 0,Y 30.902,Z 349.093,A -85,B 0,C 180,E1 -32263.025,E2 -32263.025} C_VEL
LIN {X 0,Y 31.381,Z 348.003,A -85,B 0,C 180,E1 -32261.784,E2 -32261.784} C_VEL
LIN {X 0,Y 36.834,Z 333.088,A -85,B 0,C 180,E1 -32257.641,E2 -32257.641} C_VEL
LIN {X 0,Y 38.969,Z 326.263,A -85,B 0,C 180,E1 -32257.593,E2 -32257.593} C_VEL
LIN {X 0,Y 44.905,Z 303.277,A -85,B 0,C 180,E1 -32262.368,E2 -32262.368} C_VEL
LIN {X 0,Y 46.762,Z 296.36,A -85,B 0,C 180,E1 -32262.194,E2 -32262.194} C_VEL
LIN {X 0,Y 53.587,Z 271.99,A -85,B 0,C 180,E1 -32259.406,E2 -32259.406} C_VEL
LIN {X 0,Y 54.849,Z 265.941,A -85,B 0,C 180,E1 -32265.348,E2 -32265.348} C_VEL
LIN {X 0,Y 54.79,Z 266.234,A -85,B 0,C 180,E1 -32267.869,E2 -32267.869} C_VEL
LIN {X 0,Y 54.394,Z 267.858,A -85,B 0,C 180,E1 -32269.46,E2 -32269.46} C_VEL
LIN {X 0,Y 44.022,Z 306.167,A -85,B 0,C 180,E1 -32264.253,E2 -32264.253} C_VEL
LIN {X 0,Y 44.083,Z 306.021,A -85,B 0,C 180,E1 -32263.548,E2 -32263.548} C_VEL
LIN {X 0,Y 46.762,Z 296.36,A -85,B 0,C 180,E1 -32262.194,E2 -32262.194} C_VEL
LIN {X 0,Y 50.374,Z 296.943,A -85,B 0,C 180,E1 -32260.418,E2 -32260.418} C_VEL
LIN {X 0,Y 50.374,Z 600,A -85,B 0,C 180,E1 -32260.418,E2 -32260.418} C_VEL
LIN {X 0,Y 50.374,Z 600,A -85,B 0,C 180,E1 -32260.418,E2 -32260.418}

QRS_NEXT_CUT()

QRS_NEXT()
QRS_HOME()

END
